(* IEC 61131-3 sources: JaccoSigma/tempclass/Class/ST151_IntVisu, 1 file *)

(* ---- ST151_IntVisu.st ---- *)
(*!
<Class
	Name               = "ST151_IntVisu"
	Revision           = "1.0"
	RealtimeTask       = "false"
	CyclicTask         = "false"
	BackgroundTask     = "false"
	Sigmatek           = "true"
	OSInterface        = "false"
	HighPriority       = "false"
	Automatic          = "false"
	UpdateMode         = "Prescan"
	SharedCommandTable = "true"
	Objectsize         = "(780,180)">
	<Channels>
		<Server Name="ActFreqLimitDec16to32" Visualized="true" Initialize="false" WriteProtected="false" Retentive="false" Comment="This is the actual decrease limit set to decrease server of ST151 modul.&#13;&#10;Set Frequency stepping mode limit if frequence is decreased.&#13;&#10;If the value is changed, it is transferred asynchronously to the module.&#13;&#10;If value is set to 0 the limit is automatically set."/>
		<Server Name="ActFreqLimitDec1to2" Visualized="true" Initialize="false" WriteProtected="false" Retentive="false" Comment="This is the actual decrease limit set to decrease server of ST151 modul.&#13;&#10;Set Frequency stepping mode limit if frequence is decreased.&#13;&#10;If the value is changed, it is transferred asynchronously to the module.&#13;&#10;If value is set to 0 the limit is automatically set."/>
		<Server Name="ActFreqLimitDec2to4" Visualized="true" Initialize="false" WriteProtected="false" Retentive="false" Comment="This is the actual decrease limit set to decrease server of ST151 modul.&#13;&#10;Set Frequency stepping mode limit if frequence is decreased.&#13;&#10;If the value is changed, it is transferred asynchronously to the module.&#13;&#10;If value is set to 0 the limit is automatically set."/>
		<Server Name="ActFreqLimitDec32to64" Visualized="true" Initialize="false" WriteProtected="false" Retentive="false" Comment="This is the actual decrease limit set to decrease server of ST151 modul.&#13;&#10;Set Frequency stepping mode limit if frequence is decreased.&#13;&#10;If the value is changed, it is transferred asynchronously to the module.&#13;&#10;If value is set to 0 the limit is automatically set."/>
		<Server Name="ActFreqLimitDec4to8" Visualized="true" Initialize="false" WriteProtected="false" Retentive="false" Comment="This is the actual decrease limit set to decrease server of ST151 modul.&#13;&#10;Set Frequency stepping mode limit if frequence is decreased.&#13;&#10;If the value is changed, it is transferred asynchronously to the module.&#13;&#10;If value is set to 0 the limit is automatically set."/>
		<Server Name="ActFreqLimitDec8to16" Visualized="true" Initialize="false" WriteProtected="false" Retentive="false" Comment="This is the actual decrease limit set to decrease server of ST151 modul.&#13;&#10;Set Frequency stepping mode limit if frequence is decreased.&#13;&#10;If the value is changed, it is transferred asynchronously to the module.&#13;&#10;If value is set to 0 the limit is automatically set."/>
		<Server Name="ActFreqLimitInc16to8" Visualized="true" Initialize="false" WriteProtected="false" Retentive="false" Comment="This is the actual increase limit set to ST151 modul.&#13;&#10;Set Frequency stepping mode limit if frequence is decreased.&#13;&#10;If the value is changed, it is transferred asynchronously to the module.&#13;&#10;If value is set to 0 the limit is automatically set."/>
		<Server Name="ActFreqLimitInc2to1" Visualized="true" Initialize="false" WriteProtected="false" Retentive="false" Comment="This is the actual increase limit set to ST151 modul.&#13;&#10;Set Frequency stepping mode limit if frequence is decreased.&#13;&#10;If the value is changed, it is transferred asynchronously to the module.&#13;&#10;If value is set to 0 the limit is automatically set."/>
		<Server Name="ActFreqLimitInc32to16" Visualized="true" Initialize="false" WriteProtected="false" Retentive="false" Comment="This is the actual increase limit set to ST151 modul.&#13;&#10;Set Frequency stepping mode limit if frequence is decreased.&#13;&#10;If the value is changed, it is transferred asynchronously to the module.&#13;&#10;If value is set to 0 the limit is automatically set."/>
		<Server Name="ActFreqLimitInc4to2" Visualized="true" Initialize="false" WriteProtected="false" Retentive="false" Comment="This is the actual increase limit set to ST151 modul.&#13;&#10;Set Frequency stepping mode limit if frequence is decreased.&#13;&#10;If the value is changed, it is transferred asynchronously to the module.&#13;&#10;If value is set to 0 the limit is automatically set."/>
		<Server Name="ActFreqLimitInc64to32" Visualized="true" Initialize="false" WriteProtected="false" Retentive="false" Comment="This is the actual increase limit set to ST151 modul.&#13;&#10;Set Frequency stepping mode limit if frequence is decreased.&#13;&#10;If the value is changed, it is transferred asynchronously to the module.&#13;&#10;If value is set to 0 the limit is automatically set."/>
		<Server Name="ActFreqLimitInc8to4" Visualized="true" Initialize="false" WriteProtected="false" Retentive="false" Comment="This is the actual increase limit set to ST151 modul.&#13;&#10;Set Frequency stepping mode limit if frequence is decreased.&#13;&#10;If the value is changed, it is transferred asynchronously to the module.&#13;&#10;If value is set to 0 the limit is automatically set."/>
		<Server Name="ClassSvr" Visualized="false" Initialize="false" WriteProtected="true" Retentive="false"/>
		<Server Name="CompModeSwitch" Visualized="true" Initialize="false" WriteProtected="true" Retentive="false" Comment="Shows if compatibilty mode is activated.&#13;&#10;1 .. 64 mode&#13;&#10;2 .. 32 mode"/>
		<Server Name="EnableSteps" Visualized="true" Initialize="false" WriteProtected="false" Retentive="false" Comment="Enable Steps for VOV.&#13;&#10;Enable or disable microstepping modes. The full step mode cannot be deactivated.&#13;&#10;Bit1 .. Fullstep mode&#13;&#10;Bit2 .. Halfstep mode&#13;&#10;Bit3 .. Microstepping mode 4&#13;&#10;Bit4 .. Microstepping mode 8&#13;&#10;Bit5 .. Microstepping mode 16&#13;&#10;Bit6 .. Microstepping mode 32&#13;&#10;Bit7 .. Microstepping mode 64"/>
		<Server Name="RealDec16to32" Visualized="true" Initialize="false" WriteProtected="true" Retentive="false" Comment="This is the actual decrease limit set to ST151 modul."/>
		<Server Name="RealDec1to2" Visualized="true" Initialize="false" WriteProtected="true" Retentive="false" Comment="This is the actual decrease limit set to ST151 modul."/>
		<Server Name="RealDec2to4" Visualized="true" Initialize="false" WriteProtected="true" Retentive="false" Comment="This is the actual decrease limit set to ST151 modul."/>
		<Server Name="RealDec32to64" Visualized="true" Initialize="false" WriteProtected="true" Retentive="false" Comment="This is the actual decrease limit set to ST151 modul."/>
		<Server Name="RealDec4to8" Visualized="true" Initialize="false" WriteProtected="true" Retentive="false" Comment="This is the actual decrease limit set to ST151 modul."/>
		<Server Name="RealDec8to16" Visualized="true" Initialize="false" WriteProtected="true" Retentive="false" Comment="This is the actual decrease limit set to ST151 modul."/>
		<Server Name="UpperFrequ" Visualized="true" Initialize="false" WriteProtected="false" Retentive="false" Comment="Virtuell upper frequency limit for Fullstep mode."/>
		<Server Name="VisuSchemeSwitch" Visualized="true" Initialize="false" WriteProtected="false" Retentive="false" Comment="Switch the object scheme of VOV."/>
		<Client Name="toST151Base" Required="true" Internal="false" Comment="connect to ST151Base class."/>
	</Channels>
	<RevDoku>
		<Owner Company="Sigmatek" Author="PieSte"/>
		<Dokumentation Revision="1.0" Date="22.11.2017" Author="ZoePat" Company="Sigmatek" Description="first release version."/>
	</RevDoku>
</Class>
*)
ST151_IntVisu : CLASS
  //Servers:
	ClassSvr 	: SvrChCmd_DINT;
	VisuSchemeSwitch 	: SvrCh_DINT;
	CompModeSwitch 	: SvrCh_UDINT;
	EnableSteps 	: SvrCh_bd_EnabledFreqLimit_PTofCls_ST151Base;
	UpperFrequ 	: SvrCh_UDINT;
	ActFreqLimitDec1to2 	: SvrCh_UDINT;
	ActFreqLimitDec2to4 	: SvrCh_UDINT;
	ActFreqLimitDec4to8 	: SvrCh_UDINT;
	ActFreqLimitDec8to16 	: SvrCh_UDINT;
	ActFreqLimitDec16to32 	: SvrCh_UDINT;
	ActFreqLimitDec32to64 	: SvrCh_UDINT;
	RealDec1to2 	: SvrCh_UDINT;
	RealDec2to4 	: SvrCh_UDINT;
	RealDec4to8 	: SvrCh_UDINT;
	RealDec8to16 	: SvrCh_UDINT;
	RealDec16to32 	: SvrCh_UDINT;
	RealDec32to64 	: SvrCh_UDINT;
	ActFreqLimitInc2to1 	: SvrCh_UDINT;
	ActFreqLimitInc4to2 	: SvrCh_UDINT;
	ActFreqLimitInc8to4 	: SvrCh_UDINT;
	ActFreqLimitInc16to8 	: SvrCh_UDINT;
	ActFreqLimitInc32to16 	: SvrCh_UDINT;
	ActFreqLimitInc64to32 	: SvrCh_UDINT;
  //Clients:
	toST151Base 	: CltChCmd_ST151Base;
  //Variables:
		aLastLimitsDecrease : ARRAY [0..5] OF UDINT;

  //Functions:

	FUNCTION VIRTUAL GLOBAL Init;

	FUNCTION VIRTUAL GLOBAL VisuSchemeSwitch::Write
		VAR_INPUT
			input (EAX) 	: DINT;
		END_VAR
		VAR_OUTPUT
			result (EAX) 	: DINT;
		END_VAR;

	FUNCTION VIRTUAL GLOBAL EnableSteps::Read
		VAR_OUTPUT
			output (EAX) 	: ST151Base::bd_EnabledFreqLimit;
		END_VAR;

	FUNCTION VIRTUAL GLOBAL EnableSteps::Write
		VAR_INPUT
			input (EAX) 	: ST151Base::bd_EnabledFreqLimit;
		END_VAR
		VAR_OUTPUT
			result (EAX) 	: ST151Base::bd_EnabledFreqLimit;
		END_VAR;

	FUNCTION VIRTUAL GLOBAL ActFreqLimitDec1to2::Read
		VAR_OUTPUT
			output (EAX) 	: UDINT;
		END_VAR;

	FUNCTION VIRTUAL GLOBAL ActFreqLimitDec1to2::Write
		VAR_INPUT
			input (EAX) 	: UDINT;
		END_VAR
		VAR_OUTPUT
			result (EAX) 	: UDINT;
		END_VAR;

	FUNCTION VIRTUAL GLOBAL ActFreqLimitDec2to4::Read
		VAR_OUTPUT
			output (EAX) 	: UDINT;
		END_VAR;

	FUNCTION VIRTUAL GLOBAL ActFreqLimitDec2to4::Write
		VAR_INPUT
			input (EAX) 	: UDINT;
		END_VAR
		VAR_OUTPUT
			result (EAX) 	: UDINT;
		END_VAR;

	FUNCTION VIRTUAL GLOBAL ActFreqLimitDec4to8::Read
		VAR_OUTPUT
			output (EAX) 	: UDINT;
		END_VAR;

	FUNCTION VIRTUAL GLOBAL ActFreqLimitDec4to8::Write
		VAR_INPUT
			input (EAX) 	: UDINT;
		END_VAR
		VAR_OUTPUT
			result (EAX) 	: UDINT;
		END_VAR;

	FUNCTION VIRTUAL GLOBAL ActFreqLimitDec8to16::Read
		VAR_OUTPUT
			output (EAX) 	: UDINT;
		END_VAR;

	FUNCTION VIRTUAL GLOBAL ActFreqLimitDec8to16::Write
		VAR_INPUT
			input (EAX) 	: UDINT;
		END_VAR
		VAR_OUTPUT
			result (EAX) 	: UDINT;
		END_VAR;

	FUNCTION VIRTUAL GLOBAL ActFreqLimitDec16to32::Read
		VAR_OUTPUT
			output (EAX) 	: UDINT;
		END_VAR;

	FUNCTION VIRTUAL GLOBAL ActFreqLimitDec16to32::Write
		VAR_INPUT
			input (EAX) 	: UDINT;
		END_VAR
		VAR_OUTPUT
			result (EAX) 	: UDINT;
		END_VAR;

	FUNCTION VIRTUAL GLOBAL ActFreqLimitDec32to64::Read
		VAR_OUTPUT
			output (EAX) 	: UDINT;
		END_VAR;

	FUNCTION VIRTUAL GLOBAL ActFreqLimitDec32to64::Write
		VAR_INPUT
			input (EAX) 	: UDINT;
		END_VAR
		VAR_OUTPUT
			result (EAX) 	: UDINT;
		END_VAR;

	FUNCTION VIRTUAL GLOBAL RealDec1to2::Read
		VAR_OUTPUT
			output (EAX) 	: UDINT;
		END_VAR;

	FUNCTION VIRTUAL GLOBAL RealDec2to4::Read
		VAR_OUTPUT
			output (EAX) 	: UDINT;
		END_VAR;

	FUNCTION VIRTUAL GLOBAL RealDec4to8::Read
		VAR_OUTPUT
			output (EAX) 	: UDINT;
		END_VAR;

	FUNCTION VIRTUAL GLOBAL RealDec8to16::Read
		VAR_OUTPUT
			output (EAX) 	: UDINT;
		END_VAR;

	FUNCTION VIRTUAL GLOBAL RealDec16to32::Read
		VAR_OUTPUT
			output (EAX) 	: UDINT;
		END_VAR;

	FUNCTION VIRTUAL GLOBAL RealDec32to64::Read
		VAR_OUTPUT
			output (EAX) 	: UDINT;
		END_VAR;

	FUNCTION VIRTUAL GLOBAL ActFreqLimitInc2to1::Read
		VAR_OUTPUT
			output (EAX) 	: UDINT;
		END_VAR;

	FUNCTION VIRTUAL GLOBAL ActFreqLimitInc2to1::Write
		VAR_INPUT
			input (EAX) 	: UDINT;
		END_VAR
		VAR_OUTPUT
			result (EAX) 	: UDINT;
		END_VAR;

	FUNCTION VIRTUAL GLOBAL ActFreqLimitInc4to2::Read
		VAR_OUTPUT
			output (EAX) 	: UDINT;
		END_VAR;

	FUNCTION VIRTUAL GLOBAL ActFreqLimitInc4to2::Write
		VAR_INPUT
			input (EAX) 	: UDINT;
		END_VAR
		VAR_OUTPUT
			result (EAX) 	: UDINT;
		END_VAR;

	FUNCTION VIRTUAL GLOBAL ActFreqLimitInc8to4::Read
		VAR_OUTPUT
			output (EAX) 	: UDINT;
		END_VAR;

	FUNCTION VIRTUAL GLOBAL ActFreqLimitInc8to4::Write
		VAR_INPUT
			input (EAX) 	: UDINT;
		END_VAR
		VAR_OUTPUT
			result (EAX) 	: UDINT;
		END_VAR;

	FUNCTION VIRTUAL GLOBAL ActFreqLimitInc16to8::Read
		VAR_OUTPUT
			output (EAX) 	: UDINT;
		END_VAR;

	FUNCTION VIRTUAL GLOBAL ActFreqLimitInc16to8::Write
		VAR_INPUT
			input (EAX) 	: UDINT;
		END_VAR
		VAR_OUTPUT
			result (EAX) 	: UDINT;
		END_VAR;

	FUNCTION VIRTUAL GLOBAL ActFreqLimitInc32to16::Read
		VAR_OUTPUT
			output (EAX) 	: UDINT;
		END_VAR;

	FUNCTION VIRTUAL GLOBAL ActFreqLimitInc32to16::Write
		VAR_INPUT
			input (EAX) 	: UDINT;
		END_VAR
		VAR_OUTPUT
			result (EAX) 	: UDINT;
		END_VAR;

	FUNCTION VIRTUAL GLOBAL ActFreqLimitInc64to32::Read
		VAR_OUTPUT
			output (EAX) 	: UDINT;
		END_VAR;

	FUNCTION VIRTUAL GLOBAL ActFreqLimitInc64to32::Write
		VAR_INPUT
			input (EAX) 	: UDINT;
		END_VAR
		VAR_OUTPUT
			result (EAX) 	: UDINT;
		END_VAR;
  //Tables:
	FUNCTION @STD
		VAR_OUTPUT
			ret_code	: CONFSTATES;
		END_VAR;
	FUNCTION GLOBAL TAB @CT_;
END_CLASS;

#pragma usingLtd ST151Base

FUNCTION VIRTUAL GLOBAL ST151_IntVisu::VisuSchemeSwitch::Write
	VAR_INPUT
		input (EAX) 	: DINT;
	END_VAR
	VAR_OUTPUT
		result (EAX) 	: DINT;
	END_VAR

  if input <> VisuSchemeSwitch then

    VisuSchemeSwitch := input;

    case VisuSchemeSwitch of

      //***************************************************************************************************************
      0: //simple mode
          //save last decrease limits
          aLastLimitsDecrease[0] := toST151Base.FrequLimitDecrease1to2;
          aLastLimitsDecrease[1] := toST151Base.FrequLimitDecrease2to4;
          aLastLimitsDecrease[2] := toST151Base.FrequLimitDecrease4to8;
          aLastLimitsDecrease[3] := toST151Base.FrequLimitDecrease8to16;
          aLastLimitsDecrease[4] := toST151Base.FrequLimitDecrease16to32;
          aLastLimitsDecrease[5] := toST151Base.FrequLimitDecrease32to64;
          //and set to zero for automatic calculation
          toST151Base.FrequLimitDecrease1to2.Write(input:=0);
          toST151Base.FrequLimitDecrease2to4.Write(input:=0);
          toST151Base.FrequLimitDecrease4to8.Write(input:=0);
          toST151Base.FrequLimitDecrease8to16.Write(input:=0);
          toST151Base.FrequLimitDecrease16to32.Write(input:=0);
          toST151Base.FrequLimitDecrease32to64.Write(input:=0);

      //***************************************************************************************************************
      1: //advanced mode
          toST151Base.FrequLimitDecrease1to2.Write(input:=aLastLimitsDecrease[0]);
          toST151Base.FrequLimitDecrease2to4.Write(input:=aLastLimitsDecrease[1]);
          toST151Base.FrequLimitDecrease4to8.Write(input:=aLastLimitsDecrease[2]);
          toST151Base.FrequLimitDecrease8to16.Write(input:=aLastLimitsDecrease[3]);
          toST151Base.FrequLimitDecrease16to32.Write(input:=aLastLimitsDecrease[4]);
          toST151Base.FrequLimitDecrease32to64.Write(input:=aLastLimitsDecrease[5]);

    //***************************************************************************************************************
    else

    end_case;

  end_if;

	result := VisuSchemeSwitch;

END_FUNCTION

FUNCTION VIRTUAL GLOBAL ST151_IntVisu::EnableSteps::Read
	VAR_OUTPUT
		output (EAX) 	: ST151Base::bd_EnabledFreqLimit;
	END_VAR

  EnableSteps := toST151Base.EnableSteps;
	output := EnableSteps;

END_FUNCTION

FUNCTION VIRTUAL GLOBAL ST151_IntVisu::EnableSteps::Write
	VAR_INPUT
		input (EAX) 	: ST151Base::bd_EnabledFreqLimit;
	END_VAR
	VAR_OUTPUT
		result (EAX) 	: ST151Base::bd_EnabledFreqLimit;
	END_VAR
  VAR
    mydat : UDINT;
    para  : UDINT;
  END_VAR

  mydat := EnableSteps$UDINT;
  para  := input$UDINT;

  if(para and 16#80000000) then
    if(para = 16#80000000) then
	    mydat := mydat or 16#80000000;
	  else
      mydat := mydat or (para and 16#7FFFFFFF);
    end_if;
  else
    if(para = 0) then
      mydat := mydat and 16#7FFFFFFF;
    else
	    mydat := mydat and (16#FFFFFFFF xor para);
	  end_if;
  end_if;

  toST151Base.EnableSteps.Write(input:= mydat$ST151Base::bd_EnabledFreqLimit);

	EnableSteps := mydat$ST151Base::bd_EnabledFreqLimit;

 	result := EnableSteps;

END_FUNCTION

FUNCTION VIRTUAL GLOBAL ST151_IntVisu::ActFreqLimitDec1to2::Read
	VAR_OUTPUT
		output (EAX) 	: UDINT;
	END_VAR

  ActFreqLimitDec1to2 := toST151Base.FrequLimitDecrease1to2.Read();
	output := ActFreqLimitDec1to2;

END_FUNCTION

FUNCTION VIRTUAL GLOBAL ST151_IntVisu::ActFreqLimitDec2to4::Read
	VAR_OUTPUT
		output (EAX) 	: UDINT;
	END_VAR

  ActFreqLimitDec2to4 := toST151Base.FrequLimitDecrease2to4.Read();
	output := ActFreqLimitDec2to4;

END_FUNCTION

FUNCTION VIRTUAL GLOBAL ST151_IntVisu::ActFreqLimitDec4to8::Read
	VAR_OUTPUT
		output (EAX) 	: UDINT;
	END_VAR

  ActFreqLimitDec4to8 := toST151Base.FrequLimitDecrease4to8.Read();
	output := ActFreqLimitDec4to8;

END_FUNCTION

FUNCTION VIRTUAL GLOBAL ST151_IntVisu::ActFreqLimitDec8to16::Read
	VAR_OUTPUT
		output (EAX) 	: UDINT;
	END_VAR

  ActFreqLimitDec8to16 := toST151Base.FrequLimitDecrease8to16.Read();
	output := ActFreqLimitDec8to16;

END_FUNCTION

FUNCTION VIRTUAL GLOBAL ST151_IntVisu::ActFreqLimitDec16to32::Read
	VAR_OUTPUT
		output (EAX) 	: UDINT;
	END_VAR

  ActFreqLimitDec16to32 := toST151Base.FrequLimitDecrease16to32.Read();
	output := ActFreqLimitDec16to32;

END_FUNCTION

FUNCTION VIRTUAL GLOBAL ST151_IntVisu::ActFreqLimitDec32to64::Read
	VAR_OUTPUT
		output (EAX) 	: UDINT;
	END_VAR

  ActFreqLimitDec32to64 := toST151Base.FrequLimitDecrease32to64.Read();
	output := ActFreqLimitDec32to64;

END_FUNCTION

FUNCTION VIRTUAL GLOBAL ST151_IntVisu::ActFreqLimitDec1to2::Write
	VAR_INPUT
		input (EAX) 	: UDINT;
	END_VAR
	VAR_OUTPUT
		result (EAX) 	: UDINT;
	END_VAR

	ActFreqLimitDec1to2 := input;
  toST151Base.FrequLimitDecrease1to2.Write(input:=ActFreqLimitDec1to2);
	result := ActFreqLimitDec1to2;

END_FUNCTION

FUNCTION VIRTUAL GLOBAL ST151_IntVisu::ActFreqLimitDec2to4::Write
	VAR_INPUT
		input (EAX) 	: UDINT;
	END_VAR
	VAR_OUTPUT
		result (EAX) 	: UDINT;
	END_VAR

	ActFreqLimitDec2to4 := input;
  toST151Base.FrequLimitDecrease2to4.Write(input:=ActFreqLimitDec2to4);
	result := ActFreqLimitDec2to4;

END_FUNCTION

FUNCTION VIRTUAL GLOBAL ST151_IntVisu::ActFreqLimitDec4to8::Write
	VAR_INPUT
		input (EAX) 	: UDINT;
	END_VAR
	VAR_OUTPUT
		result (EAX) 	: UDINT;
	END_VAR

	ActFreqLimitDec4to8 := input;
  toST151Base.FrequLimitDecrease4to8.Write(input:=ActFreqLimitDec4to8);
	result := ActFreqLimitDec4to8;

END_FUNCTION

FUNCTION VIRTUAL GLOBAL ST151_IntVisu::ActFreqLimitDec8to16::Write
	VAR_INPUT
		input (EAX) 	: UDINT;
	END_VAR
	VAR_OUTPUT
		result (EAX) 	: UDINT;
	END_VAR

	ActFreqLimitDec8to16 := input;
  toST151Base.FrequLimitDecrease8to16.Write(input:=ActFreqLimitDec8to16);
	result := ActFreqLimitDec8to16;

END_FUNCTION

FUNCTION VIRTUAL GLOBAL ST151_IntVisu::ActFreqLimitDec16to32::Write
	VAR_INPUT
		input (EAX) 	: UDINT;
	END_VAR
	VAR_OUTPUT
		result (EAX) 	: UDINT;
	END_VAR

	ActFreqLimitDec16to32 := input;
  toST151Base.FrequLimitDecrease16to32.Write(input:=ActFreqLimitDec16to32);
	result := ActFreqLimitDec16to32;

END_FUNCTION

FUNCTION VIRTUAL GLOBAL ST151_IntVisu::ActFreqLimitDec32to64::Write
	VAR_INPUT
		input (EAX) 	: UDINT;
	END_VAR
	VAR_OUTPUT
		result (EAX) 	: UDINT;
	END_VAR

	ActFreqLimitDec32to64 := input;
  toST151Base.FrequLimitDecrease32to64.Write(input:=ActFreqLimitDec32to64);
	result := ActFreqLimitDec32to64;

END_FUNCTION

FUNCTION VIRTUAL GLOBAL ST151_IntVisu::RealDec1to2::Read
	VAR_OUTPUT
		output (EAX) 	: UDINT;
	END_VAR

  RealDec1to2 := toST151Base.GetActFreqLimits(usValueIncDec:=1, usArrayEntry:=0, pusActCompMode:=#CompModeSwitch$USINT);
	output := RealDec1to2/CompModeSwitch;

END_FUNCTION

FUNCTION VIRTUAL GLOBAL ST151_IntVisu::RealDec2to4::Read
	VAR_OUTPUT
		output (EAX) 	: UDINT;
	END_VAR

  RealDec2to4 := toST151Base.GetActFreqLimits(usValueIncDec:=1, usArrayEntry:=1, pusActCompMode:=#CompModeSwitch$USINT);
	output := RealDec2to4/CompModeSwitch;

END_FUNCTION

FUNCTION VIRTUAL GLOBAL ST151_IntVisu::RealDec4to8::Read
	VAR_OUTPUT
		output (EAX) 	: UDINT;
	END_VAR

  RealDec4to8 := toST151Base.GetActFreqLimits(usValueIncDec:=1, usArrayEntry:=2, pusActCompMode:=#CompModeSwitch$USINT);
	output := RealDec4to8/CompModeSwitch;

END_FUNCTION

FUNCTION VIRTUAL GLOBAL ST151_IntVisu::RealDec8to16::Read
	VAR_OUTPUT
		output (EAX) 	: UDINT;
	END_VAR

  RealDec8to16 := toST151Base.GetActFreqLimits(usValueIncDec:=1, usArrayEntry:=3, pusActCompMode:=#CompModeSwitch$USINT);
	output := RealDec8to16/CompModeSwitch;

END_FUNCTION

FUNCTION VIRTUAL GLOBAL ST151_IntVisu::RealDec16to32::Read
	VAR_OUTPUT
		output (EAX) 	: UDINT;
	END_VAR

  RealDec16to32 := toST151Base.GetActFreqLimits(usValueIncDec:=1, usArrayEntry:=4, pusActCompMode:=#CompModeSwitch$USINT);
	output := RealDec16to32/CompModeSwitch;

END_FUNCTION

FUNCTION VIRTUAL GLOBAL ST151_IntVisu::RealDec32to64::Read
	VAR_OUTPUT
		output (EAX) 	: UDINT;
	END_VAR

  RealDec32to64 := toST151Base.GetActFreqLimits(usValueIncDec:=1, usArrayEntry:=5, pusActCompMode:=#CompModeSwitch$USINT);
	output := RealDec32to64/CompModeSwitch;

END_FUNCTION

FUNCTION VIRTUAL GLOBAL ST151_IntVisu::ActFreqLimitInc2to1::Write
	VAR_INPUT
		input (EAX) 	: UDINT;
	END_VAR
	VAR_OUTPUT
		result (EAX) 	: UDINT;
	END_VAR

	ActFreqLimitInc2to1 := input;
  toST151Base.FrequLimitIncrease2to1.Write(input:=ActFreqLimitInc2to1);
	result := ActFreqLimitInc2to1;

END_FUNCTION

FUNCTION VIRTUAL GLOBAL ST151_IntVisu::ActFreqLimitInc4to2::Write
	VAR_INPUT
		input (EAX) 	: UDINT;
	END_VAR
	VAR_OUTPUT
		result (EAX) 	: UDINT;
	END_VAR

	ActFreqLimitInc4to2 := input;
  toST151Base.FrequLimitIncrease4to2.Write(input:=ActFreqLimitInc4to2);
	result := ActFreqLimitInc4to2;

END_FUNCTION

FUNCTION VIRTUAL GLOBAL ST151_IntVisu::ActFreqLimitInc8to4::Write
	VAR_INPUT
		input (EAX) 	: UDINT;
	END_VAR
	VAR_OUTPUT
		result (EAX) 	: UDINT;
	END_VAR

	ActFreqLimitInc8to4 := input;
  toST151Base.FrequLimitIncrease8to4.Write(input:=ActFreqLimitInc8to4);
	result := ActFreqLimitInc8to4;

END_FUNCTION

FUNCTION VIRTUAL GLOBAL ST151_IntVisu::ActFreqLimitInc16to8::Write
	VAR_INPUT
		input (EAX) 	: UDINT;
	END_VAR
	VAR_OUTPUT
		result (EAX) 	: UDINT;
	END_VAR

	ActFreqLimitInc16to8 := input;
  toST151Base.FrequLimitIncrease16to8.Write(input:=ActFreqLimitInc16to8);
	result := ActFreqLimitInc16to8;

END_FUNCTION

FUNCTION VIRTUAL GLOBAL ST151_IntVisu::ActFreqLimitInc32to16::Write
	VAR_INPUT
		input (EAX) 	: UDINT;
	END_VAR
	VAR_OUTPUT
		result (EAX) 	: UDINT;
	END_VAR

	ActFreqLimitInc32to16 := input;
  toST151Base.FrequLimitIncrease32to16.Write(input:=ActFreqLimitInc32to16);
	result := ActFreqLimitInc32to16;

END_FUNCTION

FUNCTION VIRTUAL GLOBAL ST151_IntVisu::ActFreqLimitInc64to32::Write
	VAR_INPUT
		input (EAX) 	: UDINT;
	END_VAR
	VAR_OUTPUT
		result (EAX) 	: UDINT;
	END_VAR

	ActFreqLimitInc64to32 := input;
  toST151Base.FrequLimitIncrease64to32.Write(input:=ActFreqLimitInc64to32);
	result := ActFreqLimitInc64to32;

END_FUNCTION

FUNCTION VIRTUAL GLOBAL ST151_IntVisu::ActFreqLimitInc2to1::Read
	VAR_OUTPUT
		output (EAX) 	: UDINT;
	END_VAR

  ActFreqLimitInc2to1 := toST151Base.FrequLimitIncrease2to1.Read();
  UpperFrequ := ActFreqLimitInc2to1 + (ActFreqLimitInc2to1/10);
	output := ActFreqLimitInc2to1;

END_FUNCTION

FUNCTION VIRTUAL GLOBAL ST151_IntVisu::ActFreqLimitInc4to2::Read
	VAR_OUTPUT
		output (EAX) 	: UDINT;
	END_VAR

  ActFreqLimitInc4to2 :=toST151Base.FrequLimitIncrease4to2.Read();
	output := ActFreqLimitInc4to2;

END_FUNCTION

FUNCTION VIRTUAL GLOBAL ST151_IntVisu::ActFreqLimitInc8to4::Read
	VAR_OUTPUT
		output (EAX) 	: UDINT;
	END_VAR

  ActFreqLimitInc8to4 := toST151Base.FrequLimitIncrease8to4.Read();
	output := ActFreqLimitInc8to4;

END_FUNCTION

FUNCTION VIRTUAL GLOBAL ST151_IntVisu::ActFreqLimitInc16to8::Read
	VAR_OUTPUT
		output (EAX) 	: UDINT;
	END_VAR

  ActFreqLimitInc16to8 := toST151Base.FrequLimitIncrease16to8.Read();
	output := ActFreqLimitInc16to8;

END_FUNCTION

FUNCTION VIRTUAL GLOBAL ST151_IntVisu::ActFreqLimitInc32to16::Read
	VAR_OUTPUT
		output (EAX) 	: UDINT;
	END_VAR

  ActFreqLimitInc32to16 := toST151Base.FrequLimitIncrease32to16.Read();
	output := ActFreqLimitInc32to16;

END_FUNCTION

FUNCTION VIRTUAL GLOBAL ST151_IntVisu::ActFreqLimitInc64to32::Read
	VAR_OUTPUT
		output (EAX) 	: UDINT;
	END_VAR

  ActFreqLimitInc64to32 :=  toST151Base.FrequLimitIncrease64to32.Read();
	output := ActFreqLimitInc64to32;

END_FUNCTION

FUNCTION VIRTUAL GLOBAL ST151_IntVisu::Init

  if _FirstScan then
    if toST151Base.FrequLimitDecrease1to2 | toST151Base.FrequLimitDecrease2to4 | toST151Base.FrequLimitDecrease4to8
    | toST151Base.FrequLimitDecrease8to16 | toST151Base.FrequLimitDecrease16to32 | toST151Base.FrequLimitDecrease32to64 then
     // if a decrease limit is set, start in advanced mode
      VisuSchemeSwitch := 1;

    end_if;
    CompModeSwitch := 1;
  end_if;

END_FUNCTION
